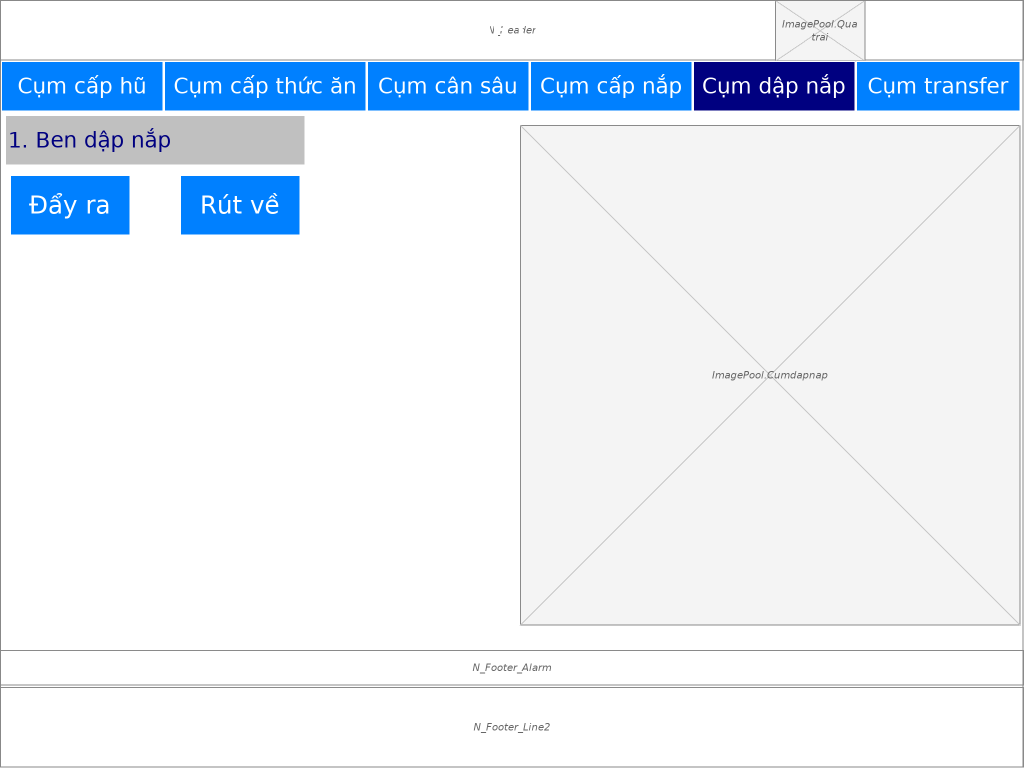
VISUALIZATION N_LidPressing2  // 1024x768
    Rectangle (180,175 120x60), "Rút về", colour toggle: PR_Line02.bCylinder_CloseLid_Retract
        OnMouseDown: execute { PR_Line02.bCylinder_CloseLid_Retract := TRUE; PR_Line02.bCylinder_CloseLid_Extend := FALSE; }
    Frame (0,687 1024x80)
        shows N_Footer_Line2()
    Frame (0,0 1024x60)
        shows N_Header()
    Textfield (353,5 400x50), "MÀN HÌNH CHẠY TAY LINE 2"
    Rectangle (10,175 120x60), "Đẩy ra", colour toggle: PR_Line02.bCylinder_CloseLid_Extend
        OnMouseDown: execute { PR_Line02.bCylinder_CloseLid_Extend := TRUE; PR_Line02.bCylinder_CloseLid_Retract := FALSE; }
    Image (775,0 90x61), input disabled if: bResetAuto1, image: ImagePool.Qua trai
        OnMouseClick: change screen: N_LidPressing1
        OnMouseClick: execute { MAIN.bModeManual := TRUE; MAIN.bModeAuto := FALSE; }
    Rectangle (1,61 162x50), "Cụm cấp hũ"
        OnMouseClick: change screen: N_JarSupply2
    Rectangle (164,61 202x50), "Cụm cấp thức ăn"
        OnMouseClick: change screen: N_FoodSupply2
    Rectangle (367,61 162x50), "Cụm cân sâu"
        OnMouseClick: change screen: N_WormWeight2
    Rectangle (530,61 162x50), "Cụm cấp nắp"
        OnMouseClick: change screen: N_LidSupply2
    Rectangle (693,61 162x50), "Cụm dập nắp"
        OnMouseClick: change screen: N_LidPressing2
    Rectangle (856,61 164x50), "Cụm transfer"
        OnMouseClick: change screen: N_Tranfer2
    Image (520,125 500x500), image: ImagePool.Cumdapnap
    Rectangle (5,115 300x50), "1. Ben dập nắp"
    Frame (0,650 1024x35)
        shows N_Footer_Alarm()
END_VISUALIZATION

(* stored: Version 1.1.0.1, ProductVersion 3.1.4024.12
   Visu N_LidPressing2: Id {8dbbcdf2-457f-42b8-86d1-f5db900964f9} *)
